TYPE DUT_SEW_Para :
STRUCT
//Geschwindigkeiten	
Geschwindigkeit_schnell		:REAL; 	// schnelle Geschwindigkeit in Anwendereihneit bei 100% Override	
Geschwindigkeit_langsam		:REAL; 	// schnelle Geschwindigkeit in Anwendereihneit bei 100% Override
Speed_Hand					:REAL; 	// langsame Geschwindigkeit in Anwendereihneit bei 100% Override
Max_Override_Hand			:INT;  	// Overridebegrenzung für Handbetrieb	
//Rampen
Beschleunigung				:INT;	// Beschleunigungsrampe in Anwendereinheit
Verzoegerung				:INT;	// Verzögerungsrampe in Anwendereinheit
//Einheiten
Einheit						:INT;	// 0 = mm/s , 1 = m/min	
//Sonstiges
Drehtausch					:BOOL;	// Motordrehsinn invertieren

// Kommastellen
Kommastelle					: INT;	// 0 = keine Kommastelle, 1 = eine Stelle ...
END_STRUCT
END_TYPE

(* stored: Version 1.1.0.1
   DUT DUT_SEW_Para: Id {c372af66-92f9-498f-98d2-9293338f7442} *)
